(* CODESYS project Soru_2.project
   Title: Adsız2
   Version: 0.0.0.0
   Author: Enes

Project tree, tasks and I/O mapping:
  MyController : TM241C24T/U, Schneider Electric, order no. TM241C24T/U, version 4.0.6.18
    application Application
      task MAST (cyclic, interval 20 ms, priority 15, watchdog 100 ms x 1) calls POU
      global variables GVL
      program POU [LD]
    DI : Digital Inputs, Schneider Electric, version 4.0.6.18
        input  iwDI_IW0 : WORD  // IW0
        input  ibDI_IB1 : BYTE  // IB1
    DQ : Digital Outputs, Schneider Electric, version 4.0.6.18
        output qwDQ_QW0 : WORD  // QW0
        output qbDQ_QB1 : BYTE  // QB1
    Counters : Counters, Schneider Electric, version 4.0.6.18
    Pulse_Generators : Pulse Generators, Schneider Electric, version 4.0.6.18
    Cartridge_1 : Cartridge, Schneider Electric, version 4.0.6.18
    IO_Bus : IO bus - TM3, Schneider Electric, version 4.0.6.18
    COM_Bus : COM bus, Schneider Electric, version 4.0.6.18
    Serial_Line_1 : Serial line, Schneider Electric, version 4.0.6.18
      SoMachine_Network_Manager : SoMachine-Network Manager, Schneider Electric, version 4.0.0.2
    Serial_Line_2 : Serial line, Schneider Electric, version 4.0.6.18
      Modbus_Manager : Modbus Manager, Schneider Electric, version 4.0.0.2
*)

// MyController/Application/GVL
VAR_GLOBAL
END_VAR

// MyController/Application/POU
PROGRAM POU
VAR
	Start: BOOL;
	Stop: BOOL;
	M0: BOOL;
	Motor_1: BOOL;
	Asiri_Akim: BOOL;
	Timer1: TON;
	Motor_2: BOOL;
	Timer2: TON;
	Motor_3: BOOL;
	Timer3: TON;
	Timer4: TON;
END_VAR
VAR // added by the converter: edge detectors and wires of the graphical bodies
    _w1 : BOOL;
END_VAR

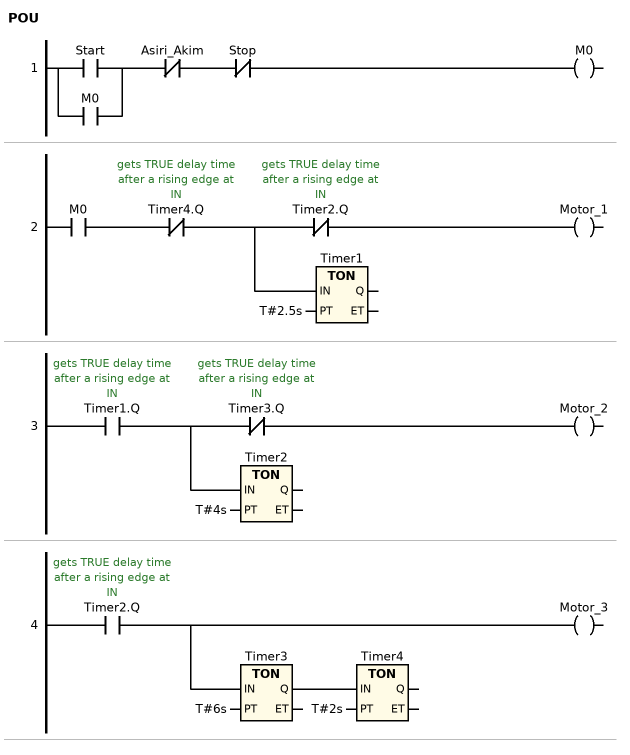
// NETWORK 1
M0 := (Start OR M0) AND NOT Asiri_Akim AND NOT Stop;

// NETWORK 2
//   Timer4.Q: gets TRUE delay time after a rising edge at IN
//   Timer2.Q: gets TRUE delay time after a rising edge at IN
_w1 := M0 AND NOT Timer4.Q;
Motor_1 := _w1 AND NOT Timer2.Q;
Timer1(IN := _w1, PT := T#2.5s); // TON

// NETWORK 3
//   Timer1.Q: gets TRUE delay time after a rising edge at IN
//   Timer3.Q: gets TRUE delay time after a rising edge at IN
Motor_2 := Timer1.Q AND NOT Timer3.Q;
Timer2(IN := Timer1.Q, PT := T#4s); // TON

// NETWORK 4
//   Timer2.Q: gets TRUE delay time after a rising edge at IN
Motor_3 := Timer2.Q;
Timer3(IN := Timer2.Q, PT := T#6s); // TON
Timer4(IN := Timer3.Q, PT := T#2s); // TON

END_PROGRAM
